(* CoDeSys 2.3 export: BUTTONEVENT.EXP *)

(* Data type in BathFB *)
TYPE ButtonEvent :
STRUCT
   (* кнопка нажата, устанавливается на один цикл *)
   downEvent:    BOOL;

   (* нажатие дольше секунды *)
   longPush:     BOOL;

   (* число, на которое надо инкрементировать, сначала 1,
   начиная с 3 секунды увеличиваеться на 1 каждую секунду *) 
   incr:         BYTE;
END_STRUCT
END_TYPE
